PROGRAM VCC2
VAR
END_VAR

END_PROGRAM

(* stored: Version 1.1.0.1, ProductVersion 3.1.4022.3
   POU VCC2: Id {4c9fc100-f02a-4673-9e05-021d5126852e}, SpecialFunc None *)
